# EPICS substitutions: pacman-softIoc/pacman_fruit.subs
file pacman_fruit.template
{ pattern
  { NAME,   VALX, VALY }
  { PACMAN,  426,  540 }
}
